FUNCTION_BLOCK FB_EmergencyStopState IMPLEMENTS I_State
VAR_INPUT
END_VAR
VAR_OUTPUT
END_VAR
VAR
	pConveyorSystem : POINTER TO FB_ConveyorSystem;
END_VAR

{warning 'add property implementation'}
PROPERTY Description : STRING
GET
END_GET
END_PROPERTY

{warning 'add method implementation '}
METHOD DetectedPartSensor1 : BOOL
END_METHOD

{warning 'add method implementation '}
METHOD DetectedPartSensor2 : BOOL
END_METHOD

{warning 'add method implementation '}
METHOD DetectedWeightSensor : BOOL
END_METHOD

METHOD FB_init : BOOL
VAR_INPUT
	bInitRetains : BOOL; // if TRUE, the retain variables are initialized (warm start / cold start)
	bInCopyCode : BOOL;  // if TRUE, the instance afterwards gets moved into the copy code (online change)
	pConveyorSystem : POINTER TO FB_ConveyorSystem;
END_VAR
THIS^.pConveyorSystem := pConveyorSystem;
END_METHOD

{warning 'add method implementation '}
METHOD PressEmergencyStop : BOOL
END_METHOD

{warning 'add method implementation '}
METHOD PressStart : BOOL
END_METHOD

{warning 'add method implementation '}
METHOD PressStop : BOOL
END_METHOD

{warning 'add method implementation '}
METHOD ProcessedWeight : BOOL
END_METHOD

END_FUNCTION_BLOCK

(* stored: Version 1.1.0.1, ProductVersion 3.1.4024.12
   POU FB_EmergencyStopState: Id {a1bac54c-0778-4a5b-afa3-ed9455949fd3}, SpecialFunc None
   Property Description: Id {6b72df5f-8153-4874-b960-0be29018c803}
   Get Get: Id {0ccb521f-e227-460c-8917-c2ba3a38535a}
   Method DetectedPartSensor1: Id {958e9a1f-fe98-42e6-a415-97876418700f}
   Method DetectedPartSensor2: Id {ac8681dd-a107-4199-8d4b-30fe5a8a1abb}
   Method DetectedWeightSensor: Id {c6ebaae1-1d64-4e60-b7a1-8071f22417b7}
   Method FB_init: Id {4e0ecc3a-6c44-4327-b565-dfa9c2e0979e}
   Method PressEmergencyStop: Id {ba1a88a6-a1e5-4980-b333-83a0e044d60e}
   Method PressStart: Id {700e1b9c-6a4e-44bc-8c67-a96fd3ea42fe}
   Method PressStop: Id {5bfdde36-5161-47c4-9e3f-9a453e460f92}
   Method ProcessedWeight: Id {8ad9570c-2171-4d47-a546-1363de7749b6} *)
